// TIA Portal V16 export
// export: Created 2022-02-28T20:47:28.6569464Z, ExportSetting WithDefaults, DisplayName Totally Integrated Automation Portal, DisplayVersion V16, DisplayName TIA Portal Version Control Interface, DisplayVersion V16, DisplayName TIA Portal Openness, DisplayVersion V16, DisplayName STEP 7 Professional, DisplayVersion V16, DisplayName STEP 7 Safety, DisplayVersion V16, DisplayName WinCC Advanced, DisplayVersion V16
VAR_GLOBAL   // PLC tag table "04_Salidas"
   MPistilos_Motor_Vdf AT %Q0.0 : Bool;   // Motor Pistilos
   MPentoflex_Motor_Logo AT %Q0.1 : Bool;   // Motor Pentoflex
END_VAR
